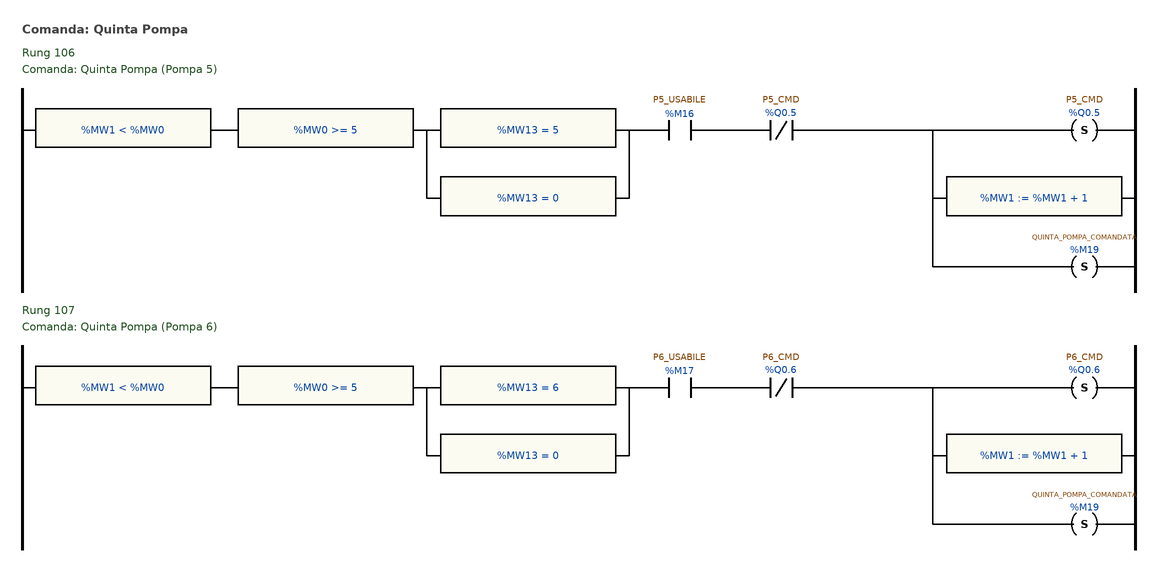

// Rung 106
// Comanda: Quinta Pompa (Pompa 5)
  LD [ %MW1 < %MW0 ]      (* NUM_POMPE_COMANDATE, NUM_POMPE_DA_COMANDARE *)
  AND [ %MW0 >= 5 ]       (* NUM_POMPE_DA_COMANDARE *)
  AND( [ %MW13 = 5 ]      (* ORDINE_QUINTA_POMPA *)
  OR [ %MW13 = 0 ]        (* ORDINE_QUINTA_POMPA *)
  )
  AND %M16                (* P5_USABILE *)
  ANDN %Q0.5              (* P5_CMD *)
  S %Q0.5                 (* P5_CMD *)
  [ %MW1 := %MW1 + 1 ]    (* NUM_POMPE_COMANDATE, NUM_POMPE_COMANDATE *)
  S %M19                  (* QUINTA_POMPA_COMANDATA *)
  // as ST:
  //   _t1 := NUM_POMPE_COMANDATE < NUM_POMPE_DA_COMANDARE AND NUM_POMPE_DA_COMANDARE >= 5 AND (ORDINE_QUINTA_POMPA = 5 OR ORDINE_QUINTA_POMPA = 0) AND P5_USABILE AND NOT P5_CMD;
  //   IF _t1 THEN P5_CMD := TRUE; END_IF;
  //   IF _t1 THEN NUM_POMPE_COMANDATE := NUM_POMPE_COMANDATE + 1; END_IF;
  //   IF _t1 THEN QUINTA_POMPA_COMANDATA := TRUE; END_IF;

// Rung 107
// Comanda: Quinta Pompa (Pompa 6)
  LD [ %MW1 < %MW0 ]      (* NUM_POMPE_COMANDATE, NUM_POMPE_DA_COMANDARE *)
  AND [ %MW0 >= 5 ]       (* NUM_POMPE_DA_COMANDARE *)
  AND( [ %MW13 = 6 ]      (* ORDINE_QUINTA_POMPA *)
  OR [ %MW13 = 0 ]        (* ORDINE_QUINTA_POMPA *)
  )
  AND %M17                (* P6_USABILE *)
  ANDN %Q0.6              (* P6_CMD *)
  S %Q0.6                 (* P6_CMD *)
  [ %MW1 := %MW1 + 1 ]    (* NUM_POMPE_COMANDATE, NUM_POMPE_COMANDATE *)
  S %M19                  (* QUINTA_POMPA_COMANDATA *)
  // as ST:
  //   _t1 := NUM_POMPE_COMANDATE < NUM_POMPE_DA_COMANDARE AND NUM_POMPE_DA_COMANDARE >= 5 AND (ORDINE_QUINTA_POMPA = 6 OR ORDINE_QUINTA_POMPA = 0) AND P6_USABILE AND NOT P6_CMD;
  //   IF _t1 THEN P6_CMD := TRUE; END_IF;
  //   IF _t1 THEN NUM_POMPE_COMANDATE := NUM_POMPE_COMANDATE + 1; END_IF;
  //   IF _t1 THEN QUINTA_POMPA_COMANDATA := TRUE; END_IF;
